# EPICS substitutions: iocs/piE625-mono/db/motor.substitutions
file "db/basic_motor.db"
{
pattern
{P,                                     M,     DTYP,        PORT, ADDR, DESC,              EGU, DIR,      VELO, VBAS, ACCL, BDST, BVEL, BACC,MRES, ERES, RDBD, UEIP, PREC, DHLM, DLLM, INIT}
{"XF\:06BM\-OP\{Mono\:1\-Ax\:FPit\}",  "Mtr", "asynMotor", PI1,  0,    "Mono Fine Pitch", um,  Pos,      1,   0.,   1.,   0,    1,    .2,   1e-3, 1e-3, 1e-3, 1, 3,    0,    0,    ""}
{"XF\:06BM\-OP\{Mono\:1\-Ax\:FRoll\}", "Mtr", "asynMotor", PI1,  1,    "Mono Fine Roll",  um,  Pos,      1,   0.,   1.,   0,    1,    .2,   1e-3, 1e-3, 1e-3, 1, 3,    0,    0,    ""}
}
